TYPE T_CHM_Filename : T_MaxString;
END_TYPE

(* stored: Version 1.1.0.1
   DUT T_CHM_Filename: Id {af99174e-08e6-47c7-8f08-6cd9da15e198} *)
